PROGRAM CncMFunctions
VAR

END_VAR

(* ========================================================= *)
(*    FUN: CncMFunctions                                     *)
(* --------------------------------------------------------- *)
(*   Desc:                                                   *)
(* Author: MK                                                *)
(*   Date: 21.12.2011                                        *)
(*   Rev.: 1.0                                               *)
(* ========================================================= *)

(*
IF CncSystem.Channel[1].M[40] = TRUE THEN
	CncSystem.Channel[1].M[40] := FALSE;
END_IF
*)

(* M-functions *)
IF CNCSystem.Channel[1].M[17] = TRUE THEN
	CNCSystem.Channel[1].M[17] := FALSE;
END_IF

(*IF CNCSystem.Channel[1].M[52] = TRUE THEN
	Temp_Tabuleiro_set:=CNCSystem.Channel[1].M_Argument[52];
		IF (IOs.Temp_Tabuleiro<Temp_Tabuleiro_set+100 AND IOs.Temp_Tabuleiro>Temp_Tabuleiro_set-100) OR Temp_Tabuleiro_set=0 THEN
			CNCSystem.Channel[1].M[52] := FALSE;
		END_IF
END_IF*)

END_PROGRAM

(* stored: Version 1.1.0.1, ProductVersion 3.1.4020.12
   POU CncMFunctions: Id {acafc1c7-34a0-4d9f-8013-7e055f97cee5}, SpecialFunc None *)
